// TIA Portal V17 export
// export: Created 2024-10-17T14:16:19.6748901Z, ExportSetting WithDefaults, DisplayName Totally Integrated Automation Portal, DisplayVersion V17 Update 4, DisplayName TIA Portal Openness, DisplayVersion V17 Update 4, DisplayName TIA Portal Version Control Interface, DisplayVersion V17, DisplayName SINAMICS Startdrive Advanced, DisplayVersion V17 Update2, DisplayName SINAMICS Startdrive G130, G150, S120, S150, SINAMICS MV, S210, DisplayVersion V17 Update2, DisplayName SINAMICS Startdrive G110M, G120, G120C, G120D, G120P, G115D, DisplayVersion V17 Update2, DisplayName STEP 7 Professional, DisplayVersion V17 Update 4, DisplayName STEP 7 Safety, DisplayVersion V17, DisplayName WinCC Advanced / Unified PC, DisplayVersion V17 Update 4
DATA_BLOCK "GlobalData"   // DB30136
TITLE = GlobalData
{ S7_Optimized_Access := 'TRUE' }
VERSION : 0.1
// stored: AutoNumber true, DBAccessibleFromOPCUA true, IsOnlyStoredInLoadMemory false, IsRetainMemResEnabled false, IsWriteProtectedInAS false, MemoryReserve 0
   VAR
      ProductionModeRequest : Bool;   // Rising edge: Request change to unit mode Production
      MaintenanceModeRequest : Bool;   // Rising edge: Request change to unit mode Maintenance
      ManualModeRequest : Bool;   // Rising edge: Request change to unit mode Manual
      UserMode01Request : Bool;   // Rising edge: Request change to user-defined unit mode 01
      UserMode02Request : Bool;   // Rising edge: Request change to user-defined unit mode 02
      UserMode03Request : Bool;   // Rising edge: Request change to user-defined unit mode 03
      UserMode04Request : Bool;   // Rising edge: Request change to user-defined unit mode 04
      UserMode05Request : Bool;   // Rising edge: Request change to user-defined unit mode 05
      ResetCmdRequest : Bool;   // Rising edge: Request control command Reset
      StartCmdRequest : Bool;   // Rising edge: Request control command Start
      StopCmdRequest : Bool;   // Rising edge: Request control command Stop
      HoldCmdRequest : Bool;   // Rising edge: Request control command Hold
      UnholdCmdRequest : Bool;   // Rising edge: Request control command Unhold
      SuspendCmdRequest : Bool;   // Rising edge: Request control command Suspend
      UnsuspendCmdRequest : Bool;   // Rising edge: Request control command Unsuspend
      AbortCmdRequest : Bool;   // Rising edge: Request control command Abort
      ClearCmdRequest : Bool;   // Rising edge: Request control command Clear
      CompleteCmdRequest : Bool;   // Rising edge: Request control command Complete
   END_VAR
BEGIN
END_DATA_BLOCK
